// LS Electric XG5000 project: 최종프로젝트(PLC)
// PLC LSPLC

PROGRAM NewProgram (task: 스캔 프로그램)

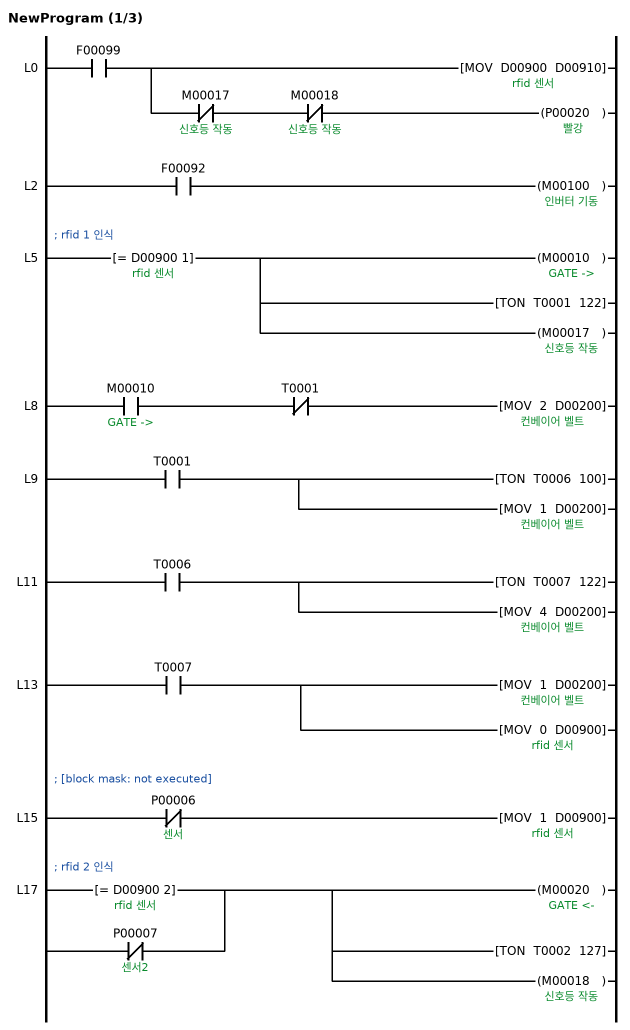
; L0
LOAD      F00099
MOV       D00900 D00910	// rfid 센서
AND NOT   M00017	// 신호등 작동
AND NOT   M00018	// 신호등 작동
OUT       P00020	// 빨강
; L2
LOAD      F00092
OUT       M00100	// 인버터 기동
// rfid 1 인식
; L5
LOAD=     D00900 1	// rfid 센서
OUT       M00010	// GATE ->
TON       T0001 122
OUT       M00017	// 신호등 작동
; L8
LOAD      M00010	// GATE ->
AND NOT   T0001
MOV       2 D00200	// 컨베이어 벨트
; L9
LOAD      T0001
TON       T0006 100
MOV       1 D00200	// 컨베이어 벨트
; L11
LOAD      T0006
TON       T0007 122
MOV       4 D00200	// 컨베이어 벨트
; L13
LOAD      T0007
MOV       1 D00200	// 컨베이어 벨트
MOV       0 D00900	// rfid 센서
; L15 (block mask: not executed)
LOAD NOT  P00006	// 센서
MOV       1 D00900	// rfid 센서
// rfid 2 인식
; L17
LOAD=     D00900 2	// rfid 센서
OR NOT    P00007	// 센서2
OUT       M00020	// GATE <-
TON       T0002 127
OUT       M00018	// 신호등 작동

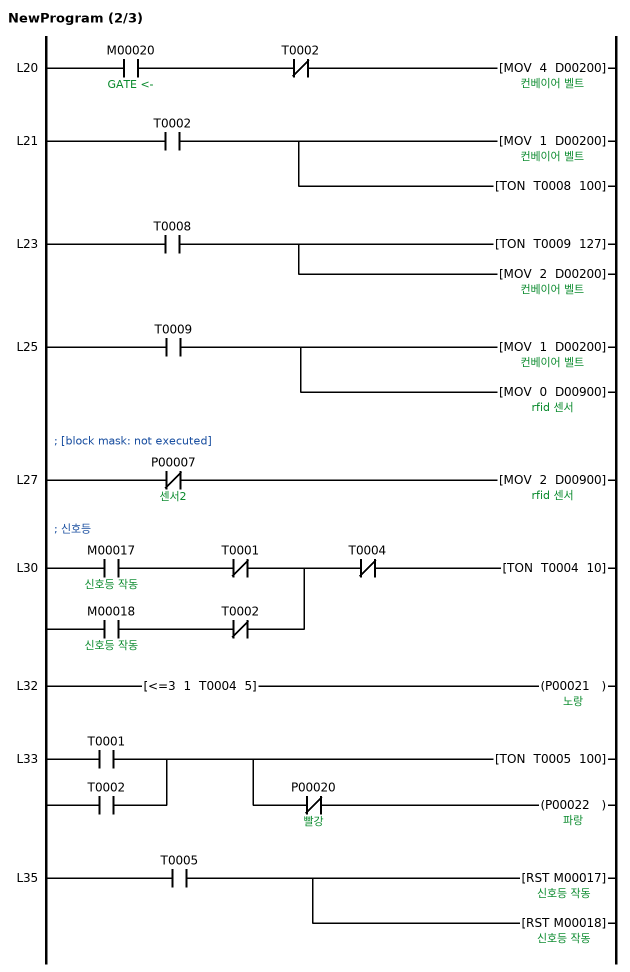
; L20
LOAD      M00020	// GATE <-
AND NOT   T0002
MOV       4 D00200	// 컨베이어 벨트
; L21
LOAD      T0002
MOV       1 D00200	// 컨베이어 벨트
TON       T0008 100
; L23
LOAD      T0008
TON       T0009 127
MOV       2 D00200	// 컨베이어 벨트
; L25
LOAD      T0009
MOV       1 D00200	// 컨베이어 벨트
MOV       0 D00900	// rfid 센서
; L27 (block mask: not executed)
LOAD NOT  P00007	// 센서2
MOV       2 D00900	// rfid 센서
// 신호등
; L30
LOAD      M00017	// 신호등 작동
AND NOT   T0001
LOAD      M00018	// 신호등 작동
AND NOT   T0002
OR LOAD
AND NOT   T0004
TON       T0004 10
; L32
LOAD<=3   1 T0004 5
OUT       P00021	// 노랑
; L33
LOAD      T0001
OR        T0002
TON       T0005 100
AND NOT   P00020	// 빨강
OUT       P00022	// 파랑
; L35
LOAD      T0005
RST       M00017	// 신호등 작동
RST       M00018	// 신호등 작동

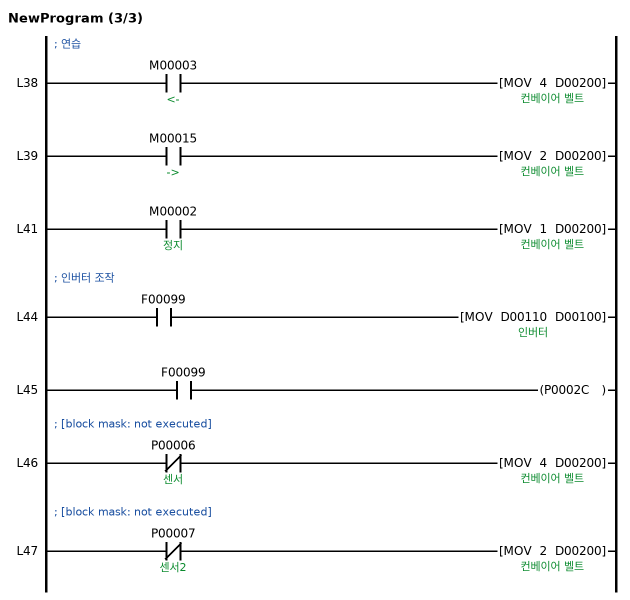
// 연습
; L38
LOAD      M00003	// <-
MOV       4 D00200	// 컨베이어 벨트
; L39
LOAD      M00015	// ->
MOV       2 D00200	// 컨베이어 벨트
; L41
LOAD      M00002	// 정지
MOV       1 D00200	// 컨베이어 벨트
// 인버터 조작
; L44
LOAD      F00099
MOV       D00110 D00100	// 인버터
; L45
LOAD      F00099
OUT       P0002C
; L46 (block mask: not executed)
LOAD NOT  P00006	// 센서
MOV       4 D00200	// 컨베이어 벨트
; L47 (block mask: not executed)
LOAD NOT  P00007	// 센서2
MOV       2 D00200	// 컨베이어 벨트